(* CODESYS project FU_sConcat7BI.xml

Project tree, tasks and I/O mapping:
  function FU_sConcat7BI [ST]
*)

// FU_sConcat7BI
//This functions combines seven strings
//This is the big input version which means any size string can be inputted, but only string variables will be accepted
//It is also faster on bigger strings
// |**Version**|**Author**| **Date** |**Changes**
// | 1         | NSN      | 05-02-19 | Creation
// | 2         | NSN      | 14-10-21 | Changed to pointer based
FUNCTION FU_sConcat7BI : STRING(255)
VAR_INPUT
	s1			:POINTER TO EASCII;			//Input String1
	s2			:POINTER TO EASCII;			//Input String2
	s3			:POINTER TO EASCII;			//Input String3
	s4			:POINTER TO EASCII;			//Input String4
	s5			:POINTER TO EASCII;			//Input String5
	s6			:POINTER TO EASCII;			//Input String6
	s7			:POINTER TO EASCII;			//Input String7
END_VAR

FU_sConcat7BIBO(sOut:=ADR(FU_sConcat7BI),s1:=s1,s2:=s2,s3:=s3,s4:=s4,s5:=s5,s6:=s6,s7:=s7,wOutSize:=255);

END_FUNCTION
